PROGRAM MAIN
VAR
	//HMI stuff
	bHMI_ForceStateVariables : BOOL := FALSE;
	stHMI_ForcedStateVariables : ST_StateVariables;
	fHMI_positionScale : LREAL; //scaling the displacement of the cart in HMI. There is probably a better way to do this.
	
	//Initialize simulator
	fInputForce : LREAL := 0.0;
	stStateVariables : ST_StateVariables;
	stInitialStateVariables : ST_StateVariables := (fX := 0.0, fXD := 0.0, fTheta := 0.000, fThetaD := 0.0);
	fbInvertedPendulum : FB_InvertedPendulum(
		fMassPendulum := 1.0, 
		fMassCart := 3.0, 
		fLengthPendulum := 0.5, 
		stInitialStateVariables := stInitialStateVariables,
		nCycleTimeMs:= 1);
		
	//Regulator
	fX_SP : LREAL := 0.0;
	fThetaSP : LREAL := 0.0;
	eRegulatorMode: E_RegulatorMode := E_RegulatorMode.eDisabled;
		
	//PID Controller for X (Outer loop)
	ePID_X_eMode : E_CTRL_MODE;
	stPID_X_settings : ST_CTRL_PID_PARAMS := (
		tCtrlCycleTime := T#10MS,
		tTaskCycleTime := T#1MS, 
		fKp := 0.2,  	 //P
		tTn := T#0MS,//I
		tTv := T#200MS,//D
		tTd := T#0MS,//Derivator filter
		fOutMaxLimit := 0.2,
		fOutMinLimit := -0.2,
		bPInTheFeedbackPath := FALSE,
		bDInTheFeedbackPath := FALSE,
		bARWOnIPartOnly := FALSE);
	fbPID_X : FB_CTRL_PID;
	
	//PID Controller for theta (Inner loop)
	ePID_Theta_eMode : E_CTRL_MODE;
	stPID_Theta_settings : ST_CTRL_PID_PARAMS := (
		tCtrlCycleTime := T#1MS, 
		tTaskCycleTime := T#1MS, 
		fKp := 200,  //P
		tTn := T#0MS,//I
		tTv := T#40MS,//D
		tTd := T#0MS,//Derivator filter
		fOutMaxLimit := 100,
		fOutMinLimit := -100,
		bPInTheFeedbackPath := FALSE,
		bDInTheFeedbackPath := FALSE,
		bARWOnIPartOnly := FALSE);
	fbPID_Theta : FB_CTRL_PID;
END_VAR

CASE eRegulatorMode OF
	E_RegulatorMode.eDisabled:
		ePID_X_eMode := E_CTRL_MODE.eCTRL_MODE_IDLE;
		ePID_Theta_eMode := E_CTRL_MODE.eCTRL_MODE_IDLE;
		
	E_RegulatorMode.ePID:
		ePID_X_eMode := E_CTRL_MODE.eCTRL_MODE_MANUAL;
		ePID_Theta_eMode := E_CTRL_MODE.eCTRL_MODE_ACTIVE;
			
	E_RegulatorMode.eCascade:
		ePID_X_eMode := E_CTRL_MODE.eCTRL_MODE_ACTIVE;
		ePID_Theta_eMode := E_CTRL_MODE.eCTRL_MODE_ACTIVE;
END_CASE

fbPID_X(
	fSetpointValue := fX_SP, 
	fActualValue := stStateVariables.fX,
	fManSyncValue := 0.0,
	eMode := ePID_X_eMode, 
	stParams := stPID_X_settings);
	fThetaSP := fbPID_X.fOut;

fbPID_Theta(
	fSetpointValue := fThetaSP, 
	fActualValue := stStateVariables.fTheta, 
	eMode := ePID_Theta_eMode, 
	stParams := stPID_Theta_settings);
	fInputForce := fbPID_Theta.fOut*-1;
	
stStateVariables := fbInvertedPendulum.Simulate(fForce := fInputForce);

IF bHMI_ForceStateVariables THEN
	fbInvertedPendulum.ForceStateVariables(stNewStateVariables := stHMI_ForcedStateVariables);
	bHMI_ForceStateVariables := FALSE;
END_IF

fHMI_positionScale := stStateVariables.fX * 200;

END_PROGRAM

(* stored: Version 1.1.0.1, ProductVersion 3.1.4024.12
   POU MAIN: Id {3ed1aa7e-7f41-4725-b882-9858b51c591a}, SpecialFunc None *)
